SUBAPPLICATION Uebung_079_AX (* Alle TECU FBs (Adapter Version) *)
  (* Standard: 61499-2; Description: Copyright (c) 2023 Meisterschulen am Ostbahnhof This program and the accompanying materials are made available under the terms of the Eclipse Public License 2.0 which is available at https://www.eclipse.org/legal/epl-2.0/ SPDX-License-Identifier: EPL-2.0 *)
  (* Version 1.0, 2026-04-19, Franz Höpfinger, Meisterschulen am Ostbahnhof, initial API and implementation (Adapter Version of Uebung_079) *)
  PACKAGE Uebungen;
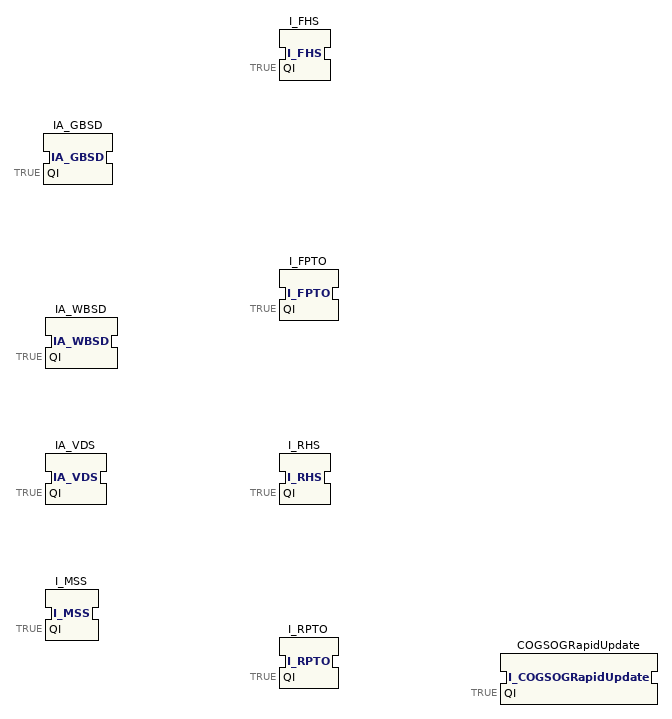
  FBS
    IA_GBSD : isobus::tecu::IA_GBSD(QI := TRUE);
    IA_VDS : isobus::tecu::IA_VDS(QI := TRUE);
    IA_WBSD : isobus::tecu::IA_WBSD(QI := TRUE);
    I_MSS : isobus::tecu::I_MSS(QI := TRUE);
    I_FHS : isobus::tecu::I_FHS(QI := TRUE);
    I_FPTO : isobus::tecu::I_FPTO(QI := TRUE);
    I_RHS : isobus::tecu::I_RHS(QI := TRUE);
    I_RPTO : isobus::tecu::I_RPTO(QI := TRUE);
    COGSOGRapidUpdate : isobus::tecu::I_COGSOGRapidUpdate(QI := TRUE);
  END_FBS
END_SUBAPPLICATION
